Fanuc KAREL source: kd00029.KL

-- PROVISIONAL review KL for V940-1; original PC SHA256 71aa7f641bf238826bedac83269228b35a2560a3dda0922f19465d51894e4d1f
-- Incomplete behavior may be omitted. Consult companion uncertainty JSON. Do not deploy.
PROGRAM KD00029
%NOLOCKGROUP
VAR
  I : INTEGER
  J : INTEGER
  B : BOOLEAN
  R : REAL
  S : STRING[80]
BEGIN
  -- V9_ZERO_TABLE_METADATA_HINT layout=0001; no indexed target words; source/name/runtime held
  -- UNRESOLVED_PC offsets 5-21; opcodes 9D,81,18,9C,12,22,9D,13,04
  -- UNRESOLVED_PC offsets 26-30; opcodes 7F
END KD00029
